TEXTLIST ErrorList2
  3 = 'Nem érkezett meg a szán a 6. hegesztéshez, vagy foglalt a hegesztő.'
  5 = 'Nem érkezett meg a 6. hegesztésnél a fej.'
  6 = 'Nem lett kész a 6. hegesztési folyamat.'
  8 = 'Nem húzódott vissza a 6. hegesztésnél a fej.'
  11 = 'Nem érkezett meg a szán a 7. hegesztéshez.'
  13 = 'Nem érkezett meg a 7. hegesztésnél a fej.'
  14 = 'Nem lett kész a 7. hegesztési folyamat.'
  16 = 'Nem húzódott vissza a 7. hegesztésnél a fej.'
  18 = 'Nem érkezett meg a szán a Kappe robotművelethez.'
  19 = 'A robot foglalt.'
  20 = 'A robot nem végzett a Kappe felrakásával.'
  22 = 'Nem érkezett meg a szán a kappézáshoz.'
  27 = 'Nem fejeződött be a kappézás művelete.'
  28 = 'Nem érkezett meg a szán a méréshez.'
  30 = 'Nem fejeződött be a mérés.'
  32 = 'Nem sikerült elküldeni a terméktípust a lézernek.'
  33 = 'Nem nyílt ki a lézer takaró.'
  34 = 'Nem sikerült elküldeni a lézernek a lézerezés parancsot.'
  36 = 'Nem záródott be a lézer takaró.'
  37 = 'Nem érkezett meg a szán a kódellenőrzéshez.'
  101 = 'Nem érkezett meg a szán a szervízboxhoz.'
  111 = 'Nem érkezett meg a szán a szervízboxhoz.'
  112 = 'Nem sikerült törölni a végmérő hibaállapotát.'
   = ''
END_TEXTLIST

(* stored: Version 1.1.0.1, ProductVersion 3.1.4020.3
   TextList ErrorList2: Id {ca07a816-f075-408e-8764-887c95dba68a} *)
